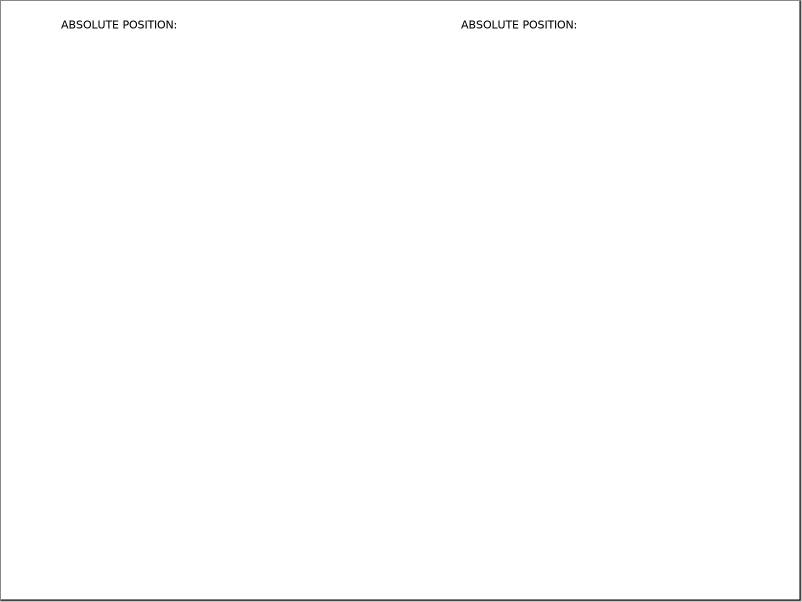
VISUALIZATION F52_Cam_In_V2  // 802x602
    Rectangle (0,0 800x600)
    Label (10,10 170x30), "ABSOLUTE POSITION:"
    Label (410,10 170x30), "ABSOLUTE POSITION:"
END_VISUALIZATION

(* stored: Version 1.1.0.1, ProductVersion 3.1.4022.7
   Visu F52_Cam_In_V2: Id {c27d756b-f594-4265-b0f0-71c1496871b7} *)
